// TIA Portal V20 export
FUNCTION "CallProductionData" : Void   // FC151, LAD
TITLE = Production data
AUTHOR : SICAR
FAMILY : ProdData
VERSION : 1.0
// Call of  FC ProductDataSimulation and LSicar Production Blocks
// stored: IsIECCheckEnabled true, SetENOAutomatically true
   // Ret_Val : Ret_Val
   VAR_TEMP   // added for the SCL form of the ladder/FBD networks
      _w1 : Bool;
      _w2 : Bool;
      _w3 : Bool;
      _w4 : Bool;
      _w5 : Bool;
      _w6 : Bool;
      _w7 : Bool;
      _w8 : Bool;
      _w9 : Bool;
      _w10 : Bool;
   END_VAR
BEGIN

REGION Network 1: BLOCK INFO HEADER
   // SIEMENS AG / (c)Copyright 2023
   // ------------------------------------------------------------------------------
   // Title:            CallProductionData(FC151)
   // Comment/Function: Call of  FC ProductDataSimulation and LSicar Production Blocks
   // Library/Family:   Automation Framework
   // Author:           Siemens Digital Industry
   // Tested with:      ---
   // Engineering:      TIA Portal V19
   // Restrictions:     -
   // Requirements:     ---
   // ------------------------------------------------------------------------------
   // Change log table:
   // Version  | Date       | Expert in charge       | Changes applied
   // ---------|------------|------------------------|------------------------------
   // 01.00.00 | 11.12.2023 | Siemens Industry Online Support
   //                         First released version
END_REGION

REGION Network 2: DESCRIPTION
   // The block is used as a calling interface for the function blocks  
   // *   _Shiftmodel
   // *   _ProdDataCycleTimer
   // *   _ProdDataCounter
   // *   _ProdDataLimitValues
   // *   _ProdDataShiftCounter
   // or
   // *   _ProdDataShiftCounterOee, ShiftProductionTimes
   // 
   // **Calling interface**  
   // The block must be called once only in the cyclic program.  
   // 
   // The block is used as a calling interface for the function blocks  
   // *   _Shiftmodel
   // *   _ProdDataCycleTimer
   // *   _ProdDataCounter
   // *   _ProdDataLimitValues
   // *   _ProdDataShiftCounter
   // or
   // *   _ProdDataShiftCounterOee, ShiftProductionTimes
   // 
   // #### Additional information
   // 
   // #### Update info
   // 
   // #### Further documentations
   // 
   // ![Icon](_Icon/reference.PNG) 
   // 
   // See:  
   // ..\Library Types\LSicar_Shiftmodel.pdf  
   // ..\Library Types\LSicar_ProdDataCycleTimer.pdf  
   // ..\Library Types\LSicar_ProdDataCounter.pdf  
   // ..\Library Types\LSicar_ProdDataLimitValues.pdf  
   // ..\Library Types\LSicar_ProdDataShiftCounter.pdf  
   // ..\Library Types\LSicar_ProdDataShiftCounterOee.pdf  
   // ..\Library Types\LSicar_ShiftProductionTimes.pdf
END_REGION

REGION Network 3
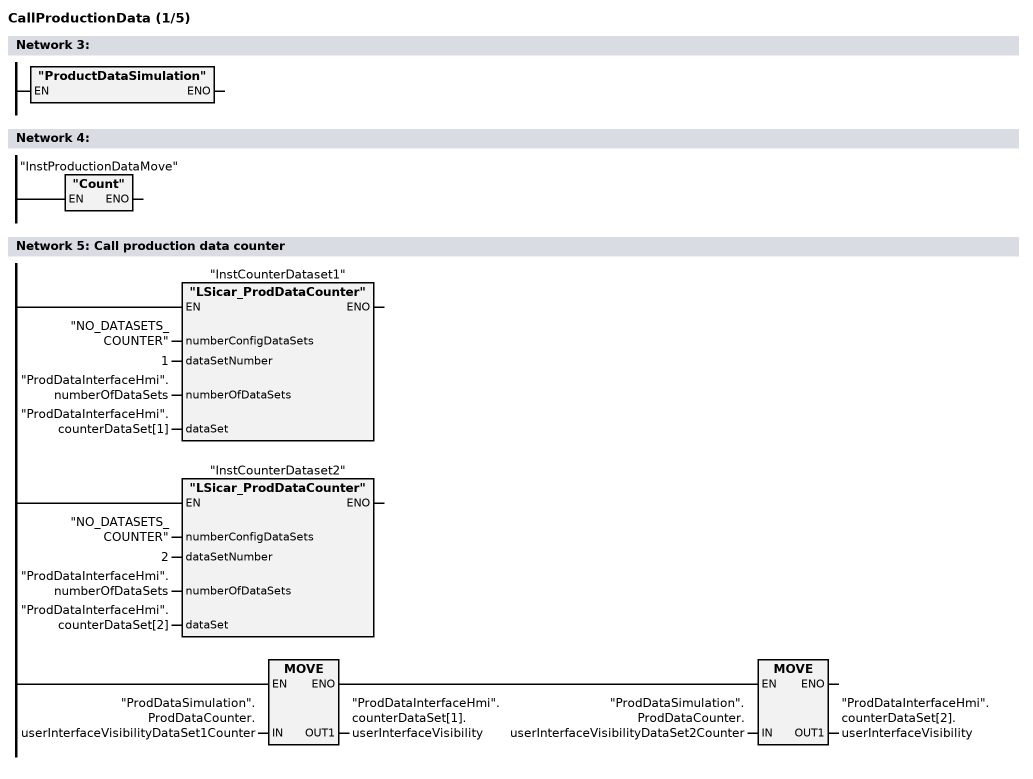
   RUNG wire#powerrail
      "ProductDataSimulation"()
   END_RUNG
   // the same network as SCL:
   "ProductDataSimulation"();
END_REGION

REGION Network 4
   RUNG wire#powerrail
      "InstProductionDataMove"()
   END_RUNG
   // the same network as SCL:
   "InstProductionDataMove"();   // "Count"
END_REGION

REGION Network 5: Call production data counter
   RUNG wire#powerrail
      "InstCounterDataset1"(numberConfigDataSets := "NO_DATASETS_COUNTER", dataSetNumber := 1, numberOfDataSets := "ProdDataInterfaceHmi".numberOfDataSets, dataSet := "ProdDataInterfaceHmi".counterDataSet[1])
   END_RUNG
   RUNG wire#powerrail
      "InstCounterDataset2"(numberConfigDataSets := "NO_DATASETS_COUNTER", dataSetNumber := 2, numberOfDataSets := "ProdDataInterfaceHmi".numberOfDataSets, dataSet := "ProdDataInterfaceHmi".counterDataSet[2])
   END_RUNG
   RUNG wire#powerrail
      Move(in := "ProdDataSimulation".ProdDataCounter.userInterfaceVisibilityDataSet1Counter, out1 => "ProdDataInterfaceHmi".counterDataSet[1].userInterfaceVisibility)
      Move(in := "ProdDataSimulation".ProdDataCounter.userInterfaceVisibilityDataSet2Counter, out1 => "ProdDataInterfaceHmi".counterDataSet[2].userInterfaceVisibility)
   END_RUNG
   // the same network as SCL:
   "InstCounterDataset1"(numberConfigDataSets := "NO_DATASETS_COUNTER",   // "LSicar_ProdDataCounter"
                         dataSetNumber := 1,
                         numberOfDataSets := "ProdDataInterfaceHmi".numberOfDataSets,
                         dataSet := "ProdDataInterfaceHmi".counterDataSet[1]);
   "InstCounterDataset2"(numberConfigDataSets := "NO_DATASETS_COUNTER",   // "LSicar_ProdDataCounter"
                         dataSetNumber := 2,
                         numberOfDataSets := "ProdDataInterfaceHmi".numberOfDataSets,
                         dataSet := "ProdDataInterfaceHmi".counterDataSet[2]);
   "ProdDataInterfaceHmi".counterDataSet[1].userInterfaceVisibility := "ProdDataSimulation".ProdDataCounter.userInterfaceVisibilityDataSet1Counter;
   "ProdDataInterfaceHmi".counterDataSet[2].userInterfaceVisibility := "ProdDataSimulation".ProdDataCounter.userInterfaceVisibilityDataSet2Counter;
END_REGION

REGION Network 6: Call production data cycle timer
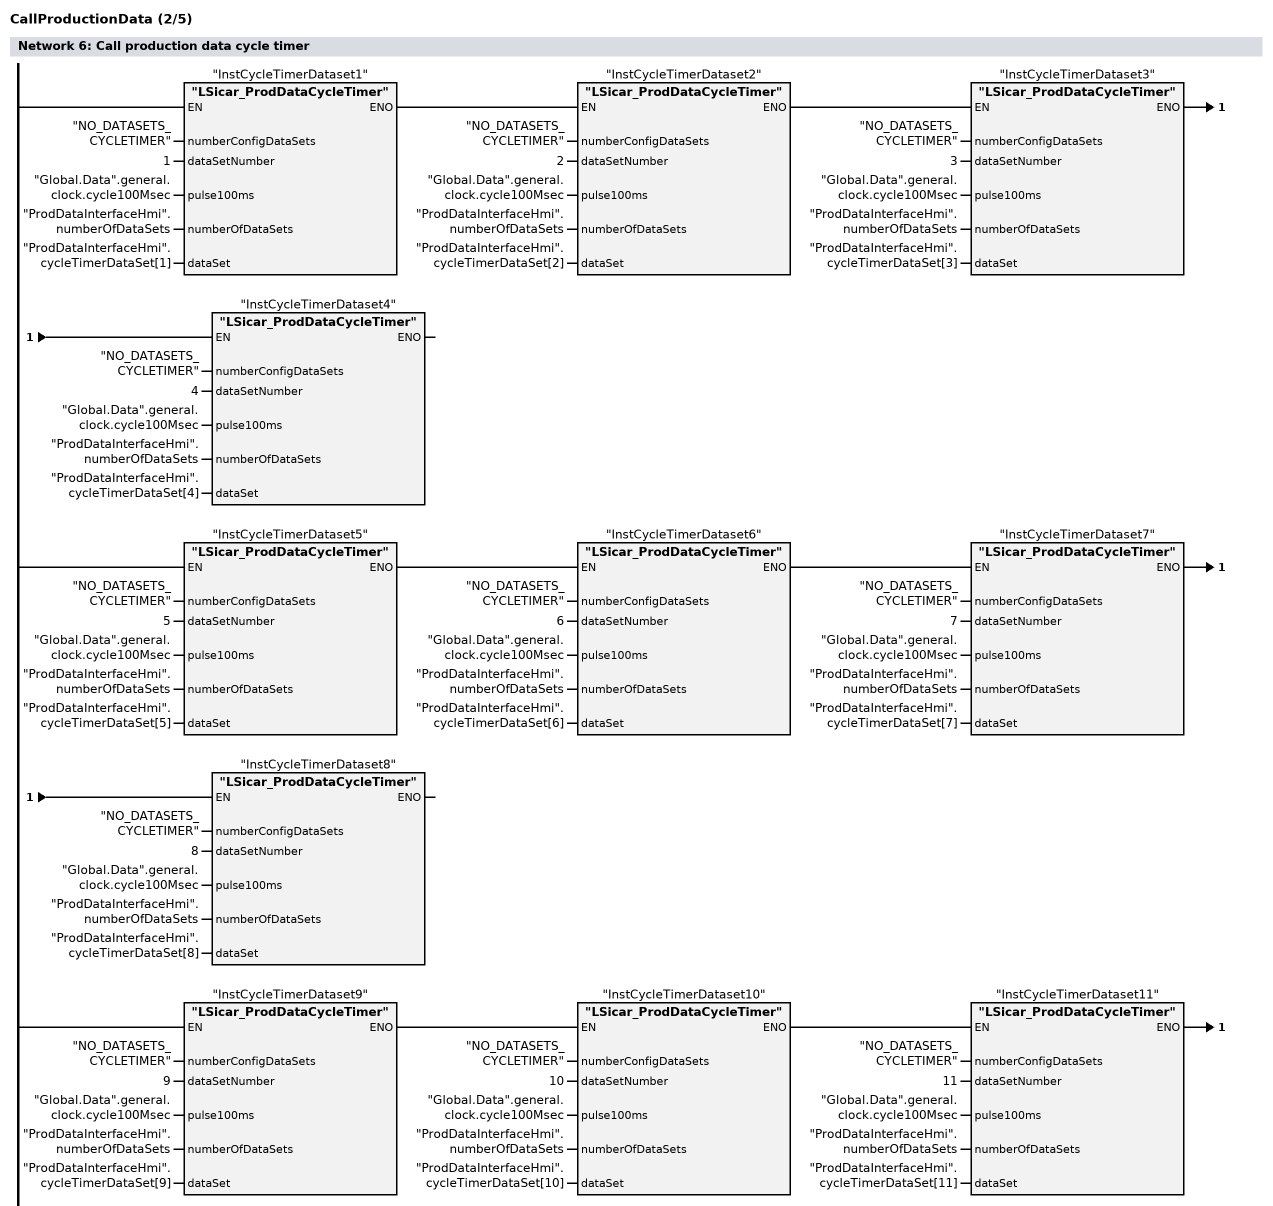
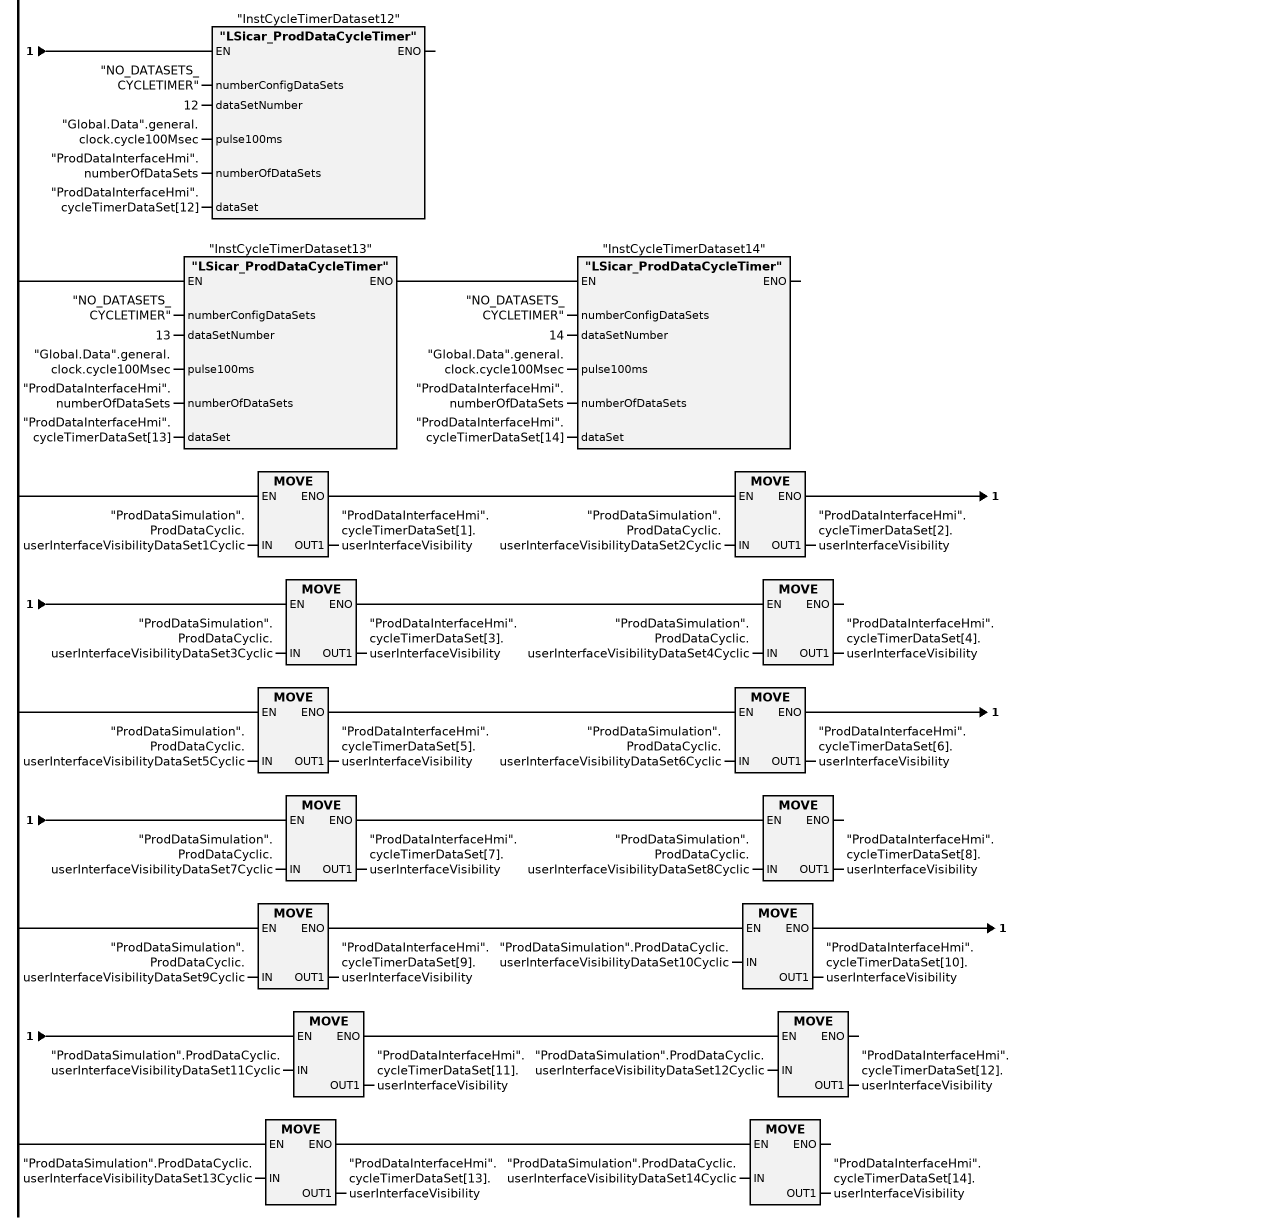
   RUNG wire#powerrail
      "InstCycleTimerDataset1"(numberConfigDataSets := "NO_DATASETS_CYCLETIMER", dataSetNumber := 1, pulse100ms := "Global.Data".general.clock.cycle100Msec, numberOfDataSets := "ProdDataInterfaceHmi".numberOfDataSets, dataSet := "ProdDataInterfaceHmi".cycleTimerDataSet[1])
      "InstCycleTimerDataset2"(numberConfigDataSets := "NO_DATASETS_CYCLETIMER", dataSetNumber := 2, pulse100ms := "Global.Data".general.clock.cycle100Msec, numberOfDataSets := "ProdDataInterfaceHmi".numberOfDataSets, dataSet := "ProdDataInterfaceHmi".cycleTimerDataSet[2])
      "InstCycleTimerDataset3"(numberConfigDataSets := "NO_DATASETS_CYCLETIMER", dataSetNumber := 3, pulse100ms := "Global.Data".general.clock.cycle100Msec, numberOfDataSets := "ProdDataInterfaceHmi".numberOfDataSets, dataSet := "ProdDataInterfaceHmi".cycleTimerDataSet[3])
      "InstCycleTimerDataset4"(numberConfigDataSets := "NO_DATASETS_CYCLETIMER", dataSetNumber := 4, pulse100ms := "Global.Data".general.clock.cycle100Msec, numberOfDataSets := "ProdDataInterfaceHmi".numberOfDataSets, dataSet := "ProdDataInterfaceHmi".cycleTimerDataSet[4])
   END_RUNG
   RUNG wire#powerrail
      "InstCycleTimerDataset5"(numberConfigDataSets := "NO_DATASETS_CYCLETIMER", dataSetNumber := 5, pulse100ms := "Global.Data".general.clock.cycle100Msec, numberOfDataSets := "ProdDataInterfaceHmi".numberOfDataSets, dataSet := "ProdDataInterfaceHmi".cycleTimerDataSet[5])
      "InstCycleTimerDataset6"(numberConfigDataSets := "NO_DATASETS_CYCLETIMER", dataSetNumber := 6, pulse100ms := "Global.Data".general.clock.cycle100Msec, numberOfDataSets := "ProdDataInterfaceHmi".numberOfDataSets, dataSet := "ProdDataInterfaceHmi".cycleTimerDataSet[6])
      "InstCycleTimerDataset7"(numberConfigDataSets := "NO_DATASETS_CYCLETIMER", dataSetNumber := 7, pulse100ms := "Global.Data".general.clock.cycle100Msec, numberOfDataSets := "ProdDataInterfaceHmi".numberOfDataSets, dataSet := "ProdDataInterfaceHmi".cycleTimerDataSet[7])
      "InstCycleTimerDataset8"(numberConfigDataSets := "NO_DATASETS_CYCLETIMER", dataSetNumber := 8, pulse100ms := "Global.Data".general.clock.cycle100Msec, numberOfDataSets := "ProdDataInterfaceHmi".numberOfDataSets, dataSet := "ProdDataInterfaceHmi".cycleTimerDataSet[8])
   END_RUNG
   RUNG wire#powerrail
      "InstCycleTimerDataset9"(numberConfigDataSets := "NO_DATASETS_CYCLETIMER", dataSetNumber := 9, pulse100ms := "Global.Data".general.clock.cycle100Msec, numberOfDataSets := "ProdDataInterfaceHmi".numberOfDataSets, dataSet := "ProdDataInterfaceHmi".cycleTimerDataSet[9])
      "InstCycleTimerDataset10"(numberConfigDataSets := "NO_DATASETS_CYCLETIMER", dataSetNumber := 10, pulse100ms := "Global.Data".general.clock.cycle100Msec, numberOfDataSets := "ProdDataInterfaceHmi".numberOfDataSets, dataSet := "ProdDataInterfaceHmi".cycleTimerDataSet[10])
      "InstCycleTimerDataset11"(numberConfigDataSets := "NO_DATASETS_CYCLETIMER", dataSetNumber := 11, pulse100ms := "Global.Data".general.clock.cycle100Msec, numberOfDataSets := "ProdDataInterfaceHmi".numberOfDataSets, dataSet := "ProdDataInterfaceHmi".cycleTimerDataSet[11])
      "InstCycleTimerDataset12"(numberConfigDataSets := "NO_DATASETS_CYCLETIMER", dataSetNumber := 12, pulse100ms := "Global.Data".general.clock.cycle100Msec, numberOfDataSets := "ProdDataInterfaceHmi".numberOfDataSets, dataSet := "ProdDataInterfaceHmi".cycleTimerDataSet[12])
   END_RUNG
   RUNG wire#powerrail
      "InstCycleTimerDataset13"(numberConfigDataSets := "NO_DATASETS_CYCLETIMER", dataSetNumber := 13, pulse100ms := "Global.Data".general.clock.cycle100Msec, numberOfDataSets := "ProdDataInterfaceHmi".numberOfDataSets, dataSet := "ProdDataInterfaceHmi".cycleTimerDataSet[13])
      "InstCycleTimerDataset14"(numberConfigDataSets := "NO_DATASETS_CYCLETIMER", dataSetNumber := 14, pulse100ms := "Global.Data".general.clock.cycle100Msec, numberOfDataSets := "ProdDataInterfaceHmi".numberOfDataSets, dataSet := "ProdDataInterfaceHmi".cycleTimerDataSet[14])
   END_RUNG
   RUNG wire#powerrail
      Move(in := "ProdDataSimulation".ProdDataCyclic.userInterfaceVisibilityDataSet1Cyclic, out1 => "ProdDataInterfaceHmi".cycleTimerDataSet[1].userInterfaceVisibility)
      Move(in := "ProdDataSimulation".ProdDataCyclic.userInterfaceVisibilityDataSet2Cyclic, out1 => "ProdDataInterfaceHmi".cycleTimerDataSet[2].userInterfaceVisibility)
      Move(in := "ProdDataSimulation".ProdDataCyclic.userInterfaceVisibilityDataSet3Cyclic, out1 => "ProdDataInterfaceHmi".cycleTimerDataSet[3].userInterfaceVisibility)
      Move(in := "ProdDataSimulation".ProdDataCyclic.userInterfaceVisibilityDataSet4Cyclic, out1 => "ProdDataInterfaceHmi".cycleTimerDataSet[4].userInterfaceVisibility)
   END_RUNG
   RUNG wire#powerrail
      Move(in := "ProdDataSimulation".ProdDataCyclic.userInterfaceVisibilityDataSet5Cyclic, out1 => "ProdDataInterfaceHmi".cycleTimerDataSet[5].userInterfaceVisibility)
      Move(in := "ProdDataSimulation".ProdDataCyclic.userInterfaceVisibilityDataSet6Cyclic, out1 => "ProdDataInterfaceHmi".cycleTimerDataSet[6].userInterfaceVisibility)
      Move(in := "ProdDataSimulation".ProdDataCyclic.userInterfaceVisibilityDataSet7Cyclic, out1 => "ProdDataInterfaceHmi".cycleTimerDataSet[7].userInterfaceVisibility)
      Move(in := "ProdDataSimulation".ProdDataCyclic.userInterfaceVisibilityDataSet8Cyclic, out1 => "ProdDataInterfaceHmi".cycleTimerDataSet[8].userInterfaceVisibility)
   END_RUNG
   RUNG wire#powerrail
      Move(in := "ProdDataSimulation".ProdDataCyclic.userInterfaceVisibilityDataSet9Cyclic, out1 => "ProdDataInterfaceHmi".cycleTimerDataSet[9].userInterfaceVisibility)
      Move(in := "ProdDataSimulation".ProdDataCyclic.userInterfaceVisibilityDataSet10Cyclic, out1 => "ProdDataInterfaceHmi".cycleTimerDataSet[10].userInterfaceVisibility)
      Move(in := "ProdDataSimulation".ProdDataCyclic.userInterfaceVisibilityDataSet11Cyclic, out1 => "ProdDataInterfaceHmi".cycleTimerDataSet[11].userInterfaceVisibility)
      Move(in := "ProdDataSimulation".ProdDataCyclic.userInterfaceVisibilityDataSet12Cyclic, out1 => "ProdDataInterfaceHmi".cycleTimerDataSet[12].userInterfaceVisibility)
   END_RUNG
   RUNG wire#powerrail
      Move(in := "ProdDataSimulation".ProdDataCyclic.userInterfaceVisibilityDataSet13Cyclic, out1 => "ProdDataInterfaceHmi".cycleTimerDataSet[13].userInterfaceVisibility)
      Move(in := "ProdDataSimulation".ProdDataCyclic.userInterfaceVisibilityDataSet14Cyclic, out1 => "ProdDataInterfaceHmi".cycleTimerDataSet[14].userInterfaceVisibility)
   END_RUNG
   // the same network as SCL:
   "InstCycleTimerDataset1"(numberConfigDataSets := "NO_DATASETS_CYCLETIMER",   // "LSicar_ProdDataCycleTimer"
                           dataSetNumber := 1,
                           pulse100ms := "Global.Data".general.clock.cycle100Msec,
                           numberOfDataSets := "ProdDataInterfaceHmi".numberOfDataSets,
                           dataSet := "ProdDataInterfaceHmi".cycleTimerDataSet[1],
                           ENO => #_w1);
   "InstCycleTimerDataset2"(EN := #_w1,   // "LSicar_ProdDataCycleTimer"
                           numberConfigDataSets := "NO_DATASETS_CYCLETIMER",
                           dataSetNumber := 2,
                           pulse100ms := "Global.Data".general.clock.cycle100Msec,
                           numberOfDataSets := "ProdDataInterfaceHmi".numberOfDataSets,
                           dataSet := "ProdDataInterfaceHmi".cycleTimerDataSet[2],
                           ENO => #_w2);
   "InstCycleTimerDataset3"(EN := #_w2,   // "LSicar_ProdDataCycleTimer"
                           numberConfigDataSets := "NO_DATASETS_CYCLETIMER",
                           dataSetNumber := 3,
                           pulse100ms := "Global.Data".general.clock.cycle100Msec,
                           numberOfDataSets := "ProdDataInterfaceHmi".numberOfDataSets,
                           dataSet := "ProdDataInterfaceHmi".cycleTimerDataSet[3],
                           ENO => #_w3);
   IF #_w3 THEN
       "InstCycleTimerDataset4"(numberConfigDataSets := "NO_DATASETS_CYCLETIMER",   // "LSicar_ProdDataCycleTimer"
                               dataSetNumber := 4,
                               pulse100ms := "Global.Data".general.clock.cycle100Msec,
                               numberOfDataSets := "ProdDataInterfaceHmi".numberOfDataSets,
                               dataSet := "ProdDataInterfaceHmi".cycleTimerDataSet[4]);
   END_IF;
   "InstCycleTimerDataset5"(numberConfigDataSets := "NO_DATASETS_CYCLETIMER",   // "LSicar_ProdDataCycleTimer"
                           dataSetNumber := 5,
                           pulse100ms := "Global.Data".general.clock.cycle100Msec,
                           numberOfDataSets := "ProdDataInterfaceHmi".numberOfDataSets,
                           dataSet := "ProdDataInterfaceHmi".cycleTimerDataSet[5],
                           ENO => #_w4);
   "InstCycleTimerDataset6"(EN := #_w4,   // "LSicar_ProdDataCycleTimer"
                           numberConfigDataSets := "NO_DATASETS_CYCLETIMER",
                           dataSetNumber := 6,
                           pulse100ms := "Global.Data".general.clock.cycle100Msec,
                           numberOfDataSets := "ProdDataInterfaceHmi".numberOfDataSets,
                           dataSet := "ProdDataInterfaceHmi".cycleTimerDataSet[6],
                           ENO => #_w5);
   "InstCycleTimerDataset7"(EN := #_w5,   // "LSicar_ProdDataCycleTimer"
                           numberConfigDataSets := "NO_DATASETS_CYCLETIMER",
                           dataSetNumber := 7,
                           pulse100ms := "Global.Data".general.clock.cycle100Msec,
                           numberOfDataSets := "ProdDataInterfaceHmi".numberOfDataSets,
                           dataSet := "ProdDataInterfaceHmi".cycleTimerDataSet[7],
                           ENO => #_w6);
   IF #_w6 THEN
       "InstCycleTimerDataset8"(numberConfigDataSets := "NO_DATASETS_CYCLETIMER",   // "LSicar_ProdDataCycleTimer"
                               dataSetNumber := 8,
                               pulse100ms := "Global.Data".general.clock.cycle100Msec,
                               numberOfDataSets := "ProdDataInterfaceHmi".numberOfDataSets,
                               dataSet := "ProdDataInterfaceHmi".cycleTimerDataSet[8]);
   END_IF;
   "InstCycleTimerDataset9"(numberConfigDataSets := "NO_DATASETS_CYCLETIMER",   // "LSicar_ProdDataCycleTimer"
                           dataSetNumber := 9,
                           pulse100ms := "Global.Data".general.clock.cycle100Msec,
                           numberOfDataSets := "ProdDataInterfaceHmi".numberOfDataSets,
                           dataSet := "ProdDataInterfaceHmi".cycleTimerDataSet[9],
                           ENO => #_w7);
   "InstCycleTimerDataset10"(EN := #_w7,   // "LSicar_ProdDataCycleTimer"
                           numberConfigDataSets := "NO_DATASETS_CYCLETIMER",
                           dataSetNumber := 10,
                           pulse100ms := "Global.Data".general.clock.cycle100Msec,
                           numberOfDataSets := "ProdDataInterfaceHmi".numberOfDataSets,
                           dataSet := "ProdDataInterfaceHmi".cycleTimerDataSet[10],
                           ENO => #_w8);
   "InstCycleTimerDataset11"(EN := #_w8,   // "LSicar_ProdDataCycleTimer"
                           numberConfigDataSets := "NO_DATASETS_CYCLETIMER",
                           dataSetNumber := 11,
                           pulse100ms := "Global.Data".general.clock.cycle100Msec,
                           numberOfDataSets := "ProdDataInterfaceHmi".numberOfDataSets,
                           dataSet := "ProdDataInterfaceHmi".cycleTimerDataSet[11],
                           ENO => #_w9);
   IF #_w9 THEN
       "InstCycleTimerDataset12"(numberConfigDataSets := "NO_DATASETS_CYCLETIMER",   // "LSicar_ProdDataCycleTimer"
                               dataSetNumber := 12,
                               pulse100ms := "Global.Data".general.clock.cycle100Msec,
                               numberOfDataSets := "ProdDataInterfaceHmi".numberOfDataSets,
                               dataSet := "ProdDataInterfaceHmi".cycleTimerDataSet[12]);
   END_IF;
   "InstCycleTimerDataset13"(numberConfigDataSets := "NO_DATASETS_CYCLETIMER",   // "LSicar_ProdDataCycleTimer"
                           dataSetNumber := 13,
                           pulse100ms := "Global.Data".general.clock.cycle100Msec,
                           numberOfDataSets := "ProdDataInterfaceHmi".numberOfDataSets,
                           dataSet := "ProdDataInterfaceHmi".cycleTimerDataSet[13],
                           ENO => #_w10);
   IF #_w10 THEN
       "InstCycleTimerDataset14"(numberConfigDataSets := "NO_DATASETS_CYCLETIMER",   // "LSicar_ProdDataCycleTimer"
                               dataSetNumber := 14,
                               pulse100ms := "Global.Data".general.clock.cycle100Msec,
                               numberOfDataSets := "ProdDataInterfaceHmi".numberOfDataSets,
                               dataSet := "ProdDataInterfaceHmi".cycleTimerDataSet[14]);
   END_IF;
   "ProdDataInterfaceHmi".cycleTimerDataSet[1].userInterfaceVisibility := "ProdDataSimulation".ProdDataCyclic.userInterfaceVisibilityDataSet1Cyclic;
   "ProdDataInterfaceHmi".cycleTimerDataSet[2].userInterfaceVisibility := "ProdDataSimulation".ProdDataCyclic.userInterfaceVisibilityDataSet2Cyclic;
   "ProdDataInterfaceHmi".cycleTimerDataSet[3].userInterfaceVisibility := "ProdDataSimulation".ProdDataCyclic.userInterfaceVisibilityDataSet3Cyclic;
   "ProdDataInterfaceHmi".cycleTimerDataSet[4].userInterfaceVisibility := "ProdDataSimulation".ProdDataCyclic.userInterfaceVisibilityDataSet4Cyclic;
   "ProdDataInterfaceHmi".cycleTimerDataSet[5].userInterfaceVisibility := "ProdDataSimulation".ProdDataCyclic.userInterfaceVisibilityDataSet5Cyclic;
   "ProdDataInterfaceHmi".cycleTimerDataSet[6].userInterfaceVisibility := "ProdDataSimulation".ProdDataCyclic.userInterfaceVisibilityDataSet6Cyclic;
   "ProdDataInterfaceHmi".cycleTimerDataSet[7].userInterfaceVisibility := "ProdDataSimulation".ProdDataCyclic.userInterfaceVisibilityDataSet7Cyclic;
   "ProdDataInterfaceHmi".cycleTimerDataSet[8].userInterfaceVisibility := "ProdDataSimulation".ProdDataCyclic.userInterfaceVisibilityDataSet8Cyclic;
   "ProdDataInterfaceHmi".cycleTimerDataSet[9].userInterfaceVisibility := "ProdDataSimulation".ProdDataCyclic.userInterfaceVisibilityDataSet9Cyclic;
   "ProdDataInterfaceHmi".cycleTimerDataSet[10].userInterfaceVisibility := "ProdDataSimulation".ProdDataCyclic.userInterfaceVisibilityDataSet10Cyclic;
   "ProdDataInterfaceHmi".cycleTimerDataSet[11].userInterfaceVisibility := "ProdDataSimulation".ProdDataCyclic.userInterfaceVisibilityDataSet11Cyclic;
   "ProdDataInterfaceHmi".cycleTimerDataSet[12].userInterfaceVisibility := "ProdDataSimulation".ProdDataCyclic.userInterfaceVisibilityDataSet12Cyclic;
   "ProdDataInterfaceHmi".cycleTimerDataSet[13].userInterfaceVisibility := "ProdDataSimulation".ProdDataCyclic.userInterfaceVisibilityDataSet13Cyclic;
   "ProdDataInterfaceHmi".cycleTimerDataSet[14].userInterfaceVisibility := "ProdDataSimulation".ProdDataCyclic.userInterfaceVisibilityDataSet14Cyclic;
END_REGION

REGION Network 7: Call production data limit values
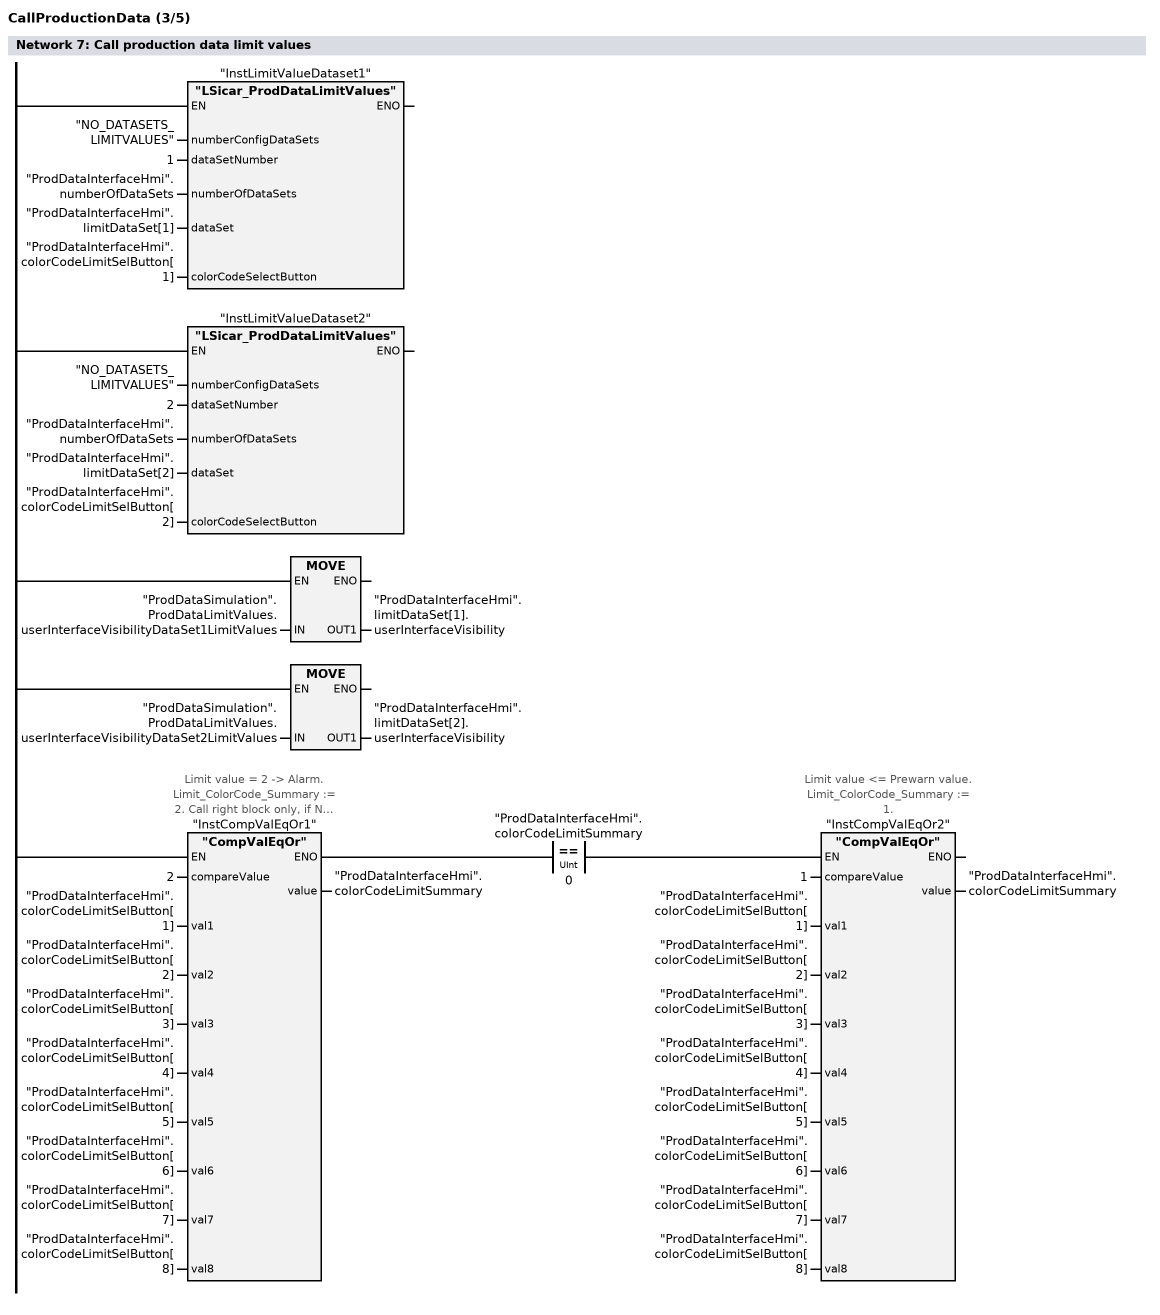
   RUNG wire#powerrail
      "InstLimitValueDataset1"(numberConfigDataSets := "NO_DATASETS_LIMITVALUES", dataSetNumber := 1, numberOfDataSets := "ProdDataInterfaceHmi".numberOfDataSets, dataSet := "ProdDataInterfaceHmi".limitDataSet[1], colorCodeSelectButton := "ProdDataInterfaceHmi".colorCodeLimitSelButton[1])
   END_RUNG
   RUNG wire#powerrail
      "InstLimitValueDataset2"(numberConfigDataSets := "NO_DATASETS_LIMITVALUES", dataSetNumber := 2, numberOfDataSets := "ProdDataInterfaceHmi".numberOfDataSets, dataSet := "ProdDataInterfaceHmi".limitDataSet[2], colorCodeSelectButton := "ProdDataInterfaceHmi".colorCodeLimitSelButton[2])
   END_RUNG
   RUNG wire#powerrail
      Move(in := "ProdDataSimulation".ProdDataLimitValues.userInterfaceVisibilityDataSet1LimitValues, out1 => "ProdDataInterfaceHmi".limitDataSet[1].userInterfaceVisibility)
   END_RUNG
   RUNG wire#powerrail
      Move(in := "ProdDataSimulation".ProdDataLimitValues.userInterfaceVisibilityDataSet2LimitValues, out1 => "ProdDataInterfaceHmi".limitDataSet[2].userInterfaceVisibility)
   END_RUNG
   RUNG wire#powerrail
      "InstCompValEqOr1"(compareValue := 2, val1 := "ProdDataInterfaceHmi".colorCodeLimitSelButton[1], val2 := "ProdDataInterfaceHmi".colorCodeLimitSelButton[2], val3 := "ProdDataInterfaceHmi".colorCodeLimitSelButton[3], val4 := "ProdDataInterfaceHmi".colorCodeLimitSelButton[4], val5 := "ProdDataInterfaceHmi".colorCodeLimitSelButton[5], val6 := "ProdDataInterfaceHmi".colorCodeLimitSelButton[6], val7 := "ProdDataInterfaceHmi".colorCodeLimitSelButton[7], val8 := "ProdDataInterfaceHmi".colorCodeLimitSelButton[8], value => "ProdDataInterfaceHmi".colorCodeLimitSummary)   // Limit value = 2 -> Alarm. Limit_ColorCode_Summary := 2. Call right block only, if NO alarm (VALUE = 0) is pending here; alarm is higher prior.
      { S7_Templates := "SrcType := UInt" } EQ_Contact(in1 := "ProdDataInterfaceHmi".colorCodeLimitSummary, in2 := 0)
      "InstCompValEqOr2"(compareValue := 1, val1 := "ProdDataInterfaceHmi".colorCodeLimitSelButton[1], val2 := "ProdDataInterfaceHmi".colorCodeLimitSelButton[2], val3 := "ProdDataInterfaceHmi".colorCodeLimitSelButton[3], val4 := "ProdDataInterfaceHmi".colorCodeLimitSelButton[4], val5 := "ProdDataInterfaceHmi".colorCodeLimitSelButton[5], val6 := "ProdDataInterfaceHmi".colorCodeLimitSelButton[6], val7 := "ProdDataInterfaceHmi".colorCodeLimitSelButton[7], val8 := "ProdDataInterfaceHmi".colorCodeLimitSelButton[8], value => "ProdDataInterfaceHmi".colorCodeLimitSummary)   // Limit value <= Prewarn value. Limit_ColorCode_Summary := 1.
   END_RUNG
   // the same network as SCL:
   "InstLimitValueDataset1"(numberConfigDataSets := "NO_DATASETS_LIMITVALUES",   // "LSicar_ProdDataLimitValues"
                           dataSetNumber := 1,
                           numberOfDataSets := "ProdDataInterfaceHmi".numberOfDataSets,
                           dataSet := "ProdDataInterfaceHmi".limitDataSet[1],
                           colorCodeSelectButton := "ProdDataInterfaceHmi".colorCodeLimitSelButton[1]);
   "InstLimitValueDataset2"(numberConfigDataSets := "NO_DATASETS_LIMITVALUES",   // "LSicar_ProdDataLimitValues"
                           dataSetNumber := 2,
                           numberOfDataSets := "ProdDataInterfaceHmi".numberOfDataSets,
                           dataSet := "ProdDataInterfaceHmi".limitDataSet[2],
                           colorCodeSelectButton := "ProdDataInterfaceHmi".colorCodeLimitSelButton[2]);
   "ProdDataInterfaceHmi".limitDataSet[1].userInterfaceVisibility := "ProdDataSimulation".ProdDataLimitValues.userInterfaceVisibilityDataSet1LimitValues;
   "ProdDataInterfaceHmi".limitDataSet[2].userInterfaceVisibility := "ProdDataSimulation".ProdDataLimitValues.userInterfaceVisibilityDataSet2LimitValues;
   "InstCompValEqOr1"(compareValue := 2,   // "CompValEqOr": Limit value = 2 -> Alarm. Limit_ColorCode_Summary := 2. Call right block only, if NO alarm (VALUE = 0) is pending here; alarm is higher prior.
                      val1 := "ProdDataInterfaceHmi".colorCodeLimitSelButton[1],
                      val2 := "ProdDataInterfaceHmi".colorCodeLimitSelButton[2],
                      val3 := "ProdDataInterfaceHmi".colorCodeLimitSelButton[3],
                      val4 := "ProdDataInterfaceHmi".colorCodeLimitSelButton[4],
                      val5 := "ProdDataInterfaceHmi".colorCodeLimitSelButton[5],
                      val6 := "ProdDataInterfaceHmi".colorCodeLimitSelButton[6],
                      val7 := "ProdDataInterfaceHmi".colorCodeLimitSelButton[7],
                      val8 := "ProdDataInterfaceHmi".colorCodeLimitSelButton[8],
                      value => "ProdDataInterfaceHmi".colorCodeLimitSummary,
                      ENO => #_w1);
   IF #_w1 AND ("ProdDataInterfaceHmi".colorCodeLimitSummary = 0) THEN
       "InstCompValEqOr2"(compareValue := 1,   // "CompValEqOr": Limit value <= Prewarn value. Limit_ColorCode_Summary := 1.
                          val1 := "ProdDataInterfaceHmi".colorCodeLimitSelButton[1],
                          val2 := "ProdDataInterfaceHmi".colorCodeLimitSelButton[2],
                          val3 := "ProdDataInterfaceHmi".colorCodeLimitSelButton[3],
                          val4 := "ProdDataInterfaceHmi".colorCodeLimitSelButton[4],
                          val5 := "ProdDataInterfaceHmi".colorCodeLimitSelButton[5],
                          val6 := "ProdDataInterfaceHmi".colorCodeLimitSelButton[6],
                          val7 := "ProdDataInterfaceHmi".colorCodeLimitSelButton[7],
                          val8 := "ProdDataInterfaceHmi".colorCodeLimitSelButton[8],
                          value => "ProdDataInterfaceHmi".colorCodeLimitSummary);
   END_IF;
END_REGION

REGION Network 8: Call production data shift counter
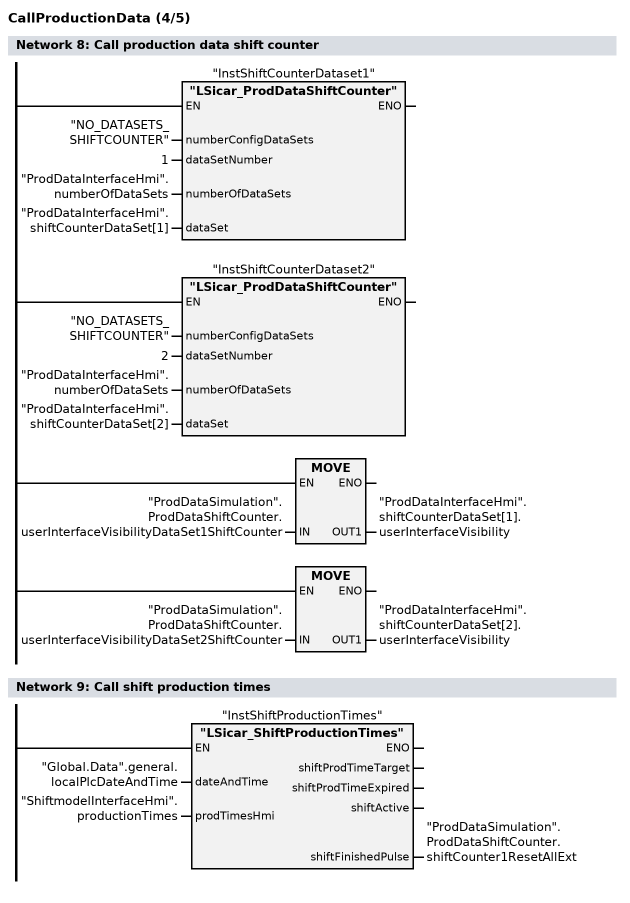
   RUNG wire#powerrail
      "InstShiftCounterDataset1"(numberConfigDataSets := "NO_DATASETS_SHIFTCOUNTER", dataSetNumber := 1, numberOfDataSets := "ProdDataInterfaceHmi".numberOfDataSets, dataSet := "ProdDataInterfaceHmi".shiftCounterDataSet[1])
   END_RUNG
   RUNG wire#powerrail
      "InstShiftCounterDataset2"(numberConfigDataSets := "NO_DATASETS_SHIFTCOUNTER", dataSetNumber := 2, numberOfDataSets := "ProdDataInterfaceHmi".numberOfDataSets, dataSet := "ProdDataInterfaceHmi".shiftCounterDataSet[2])
   END_RUNG
   RUNG wire#powerrail
      Move(in := "ProdDataSimulation".ProdDataShiftCounter.userInterfaceVisibilityDataSet1ShiftCounter, out1 => "ProdDataInterfaceHmi".shiftCounterDataSet[1].userInterfaceVisibility)
   END_RUNG
   RUNG wire#powerrail
      Move(in := "ProdDataSimulation".ProdDataShiftCounter.userInterfaceVisibilityDataSet2ShiftCounter, out1 => "ProdDataInterfaceHmi".shiftCounterDataSet[2].userInterfaceVisibility)
   END_RUNG
   // the same network as SCL:
   "InstShiftCounterDataset1"(numberConfigDataSets := "NO_DATASETS_SHIFTCOUNTER",   // "LSicar_ProdDataShiftCounter"
                           dataSetNumber := 1,
                           numberOfDataSets := "ProdDataInterfaceHmi".numberOfDataSets,
                           dataSet := "ProdDataInterfaceHmi".shiftCounterDataSet[1]);
   "InstShiftCounterDataset2"(numberConfigDataSets := "NO_DATASETS_SHIFTCOUNTER",   // "LSicar_ProdDataShiftCounter"
                           dataSetNumber := 2,
                           numberOfDataSets := "ProdDataInterfaceHmi".numberOfDataSets,
                           dataSet := "ProdDataInterfaceHmi".shiftCounterDataSet[2]);
   "ProdDataInterfaceHmi".shiftCounterDataSet[1].userInterfaceVisibility := "ProdDataSimulation".ProdDataShiftCounter.userInterfaceVisibilityDataSet1ShiftCounter;
   "ProdDataInterfaceHmi".shiftCounterDataSet[2].userInterfaceVisibility := "ProdDataSimulation".ProdDataShiftCounter.userInterfaceVisibilityDataSet2ShiftCounter;
END_REGION

REGION Network 9: Call shift production times
   RUNG wire#powerrail
      "InstShiftProductionTimes"(dateAndTime := "Global.Data".general.localPlcDateAndTime, prodTimesHmi := "ShiftmodelInterfaceHmi".productionTimes, shiftProdTimeTarget =>, shiftProdTimeExpired =>, shiftActive =>, shiftFinishedPulse => "ProdDataSimulation".ProdDataShiftCounter.shiftCounter1ResetAllExt)
   END_RUNG
   // the same network as SCL:
   "InstShiftProductionTimes"(dateAndTime := "Global.Data".general.localPlcDateAndTime,   // "LSicar_ShiftProductionTimes"
                           prodTimesHmi := "ShiftmodelInterfaceHmi".productionTimes,
                           shiftFinishedPulse => "ProdDataSimulation".ProdDataShiftCounter.shiftCounter1ResetAllExt);
END_REGION

REGION Network 10: Call production data shift counter OEE
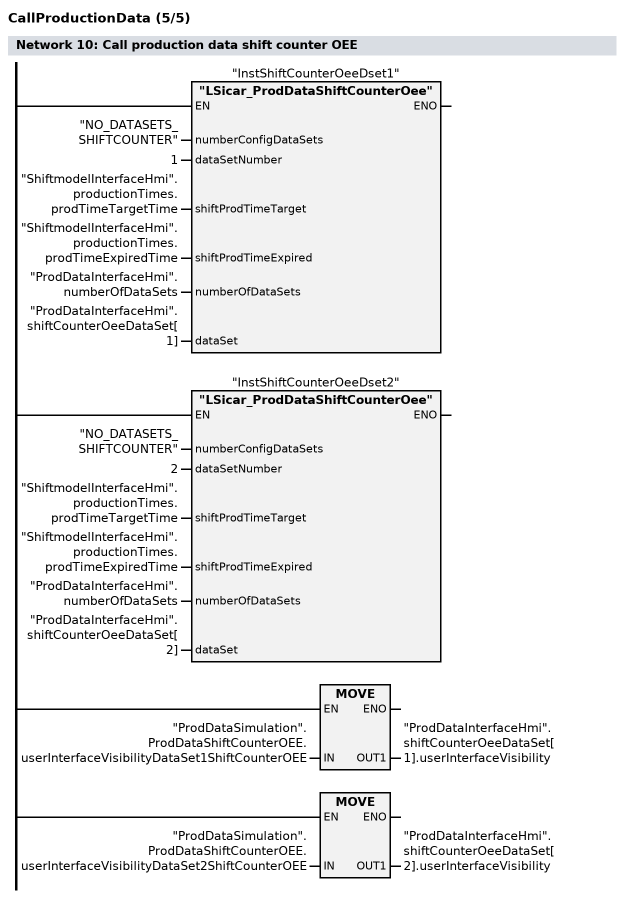
   RUNG wire#powerrail
      "InstShiftCounterOeeDset1"(numberConfigDataSets := "NO_DATASETS_SHIFTCOUNTER", dataSetNumber := 1, shiftProdTimeTarget := "ShiftmodelInterfaceHmi".productionTimes.prodTimeTargetTime, shiftProdTimeExpired := "ShiftmodelInterfaceHmi".productionTimes.prodTimeExpiredTime, numberOfDataSets := "ProdDataInterfaceHmi".numberOfDataSets, dataSet := "ProdDataInterfaceHmi".shiftCounterOeeDataSet[1])
   END_RUNG
   RUNG wire#powerrail
      "InstShiftCounterOeeDset2"(numberConfigDataSets := "NO_DATASETS_SHIFTCOUNTER", dataSetNumber := 2, shiftProdTimeTarget := "ShiftmodelInterfaceHmi".productionTimes.prodTimeTargetTime, shiftProdTimeExpired := "ShiftmodelInterfaceHmi".productionTimes.prodTimeExpiredTime, numberOfDataSets := "ProdDataInterfaceHmi".numberOfDataSets, dataSet := "ProdDataInterfaceHmi".shiftCounterOeeDataSet[2])
   END_RUNG
   RUNG wire#powerrail
      Move(in := "ProdDataSimulation".ProdDataShiftCounterOEE.userInterfaceVisibilityDataSet1ShiftCounterOEE, out1 => "ProdDataInterfaceHmi".shiftCounterOeeDataSet[1].userInterfaceVisibility)
   END_RUNG
   RUNG wire#powerrail
      Move(in := "ProdDataSimulation".ProdDataShiftCounterOEE.userInterfaceVisibilityDataSet2ShiftCounterOEE, out1 => "ProdDataInterfaceHmi".shiftCounterOeeDataSet[2].userInterfaceVisibility)
   END_RUNG
   // the same network as SCL:
   "InstShiftCounterOeeDset1"(numberConfigDataSets := "NO_DATASETS_SHIFTCOUNTER",   // "LSicar_ProdDataShiftCounterOee"
                           dataSetNumber := 1,
                           shiftProdTimeTarget := "ShiftmodelInterfaceHmi".productionTimes.prodTimeTargetTime,
                           shiftProdTimeExpired := "ShiftmodelInterfaceHmi".productionTimes.prodTimeExpiredTime,
                           numberOfDataSets := "ProdDataInterfaceHmi".numberOfDataSets,
                           dataSet := "ProdDataInterfaceHmi".shiftCounterOeeDataSet[1]);
   "InstShiftCounterOeeDset2"(numberConfigDataSets := "NO_DATASETS_SHIFTCOUNTER",   // "LSicar_ProdDataShiftCounterOee"
                           dataSetNumber := 2,
                           shiftProdTimeTarget := "ShiftmodelInterfaceHmi".productionTimes.prodTimeTargetTime,
                           shiftProdTimeExpired := "ShiftmodelInterfaceHmi".productionTimes.prodTimeExpiredTime,
                           numberOfDataSets := "ProdDataInterfaceHmi".numberOfDataSets,
                           dataSet := "ProdDataInterfaceHmi".shiftCounterOeeDataSet[2]);
   "ProdDataInterfaceHmi".shiftCounterOeeDataSet[1].userInterfaceVisibility := "ProdDataSimulation".ProdDataShiftCounterOEE.userInterfaceVisibilityDataSet1ShiftCounterOEE;
   "ProdDataInterfaceHmi".shiftCounterOeeDataSet[2].userInterfaceVisibility := "ProdDataSimulation".ProdDataShiftCounterOEE.userInterfaceVisibilityDataSet2ShiftCounterOEE;
END_REGION
END_FUNCTION
